{attribute 'linkalways'} 
{attribute 'no_explicit_call' := 'This FB is a CLASS and must be accessed using methods or properties'}
{attribute 'enable_dynamic_creation'}
FUNCTION_BLOCK FINAL MUL_INT EXTENDS Node
VAR
	in1 : _INT(0);
	in2 : _INT(0);
	out : _INT(0);
END_VAR

METHOD PUBLIC Clone : I_Node
VAR
	pNode : POINTER TO MUL_INT;
END_VAR
pNode := __NEW(MUL_INT);
Clone := pNode^;
END_METHOD

METHOD FB_init : BOOL
VAR_INPUT
	bInitRetains : BOOL; // if TRUE, the retain variables are initialized (warm start / cold start)
	bInCopyCode : BOOL;  // if TRUE, the instance afterwards gets moved into the copy code (online change)
END_VAR
AddInput('in1',THIS^.in1);
AddInput('in2',THIS^.in2);
AddOutput('out', THIS^.out);
END_METHOD

METHOD PROTECTED OnExecute
VAR
END_VAR
out.Value := in1.Value * in2.Value;
END_METHOD

END_FUNCTION_BLOCK

(* stored: Version 1.1.0.1, ProductVersion 3.1.4024.15
   POU MUL_INT: Id {147e88f2-4c59-4cc2-a2c0-754993355c72}, SpecialFunc None
   Folder Constructor: Id {3311f08b-3fa3-4e51-8756-cc330fadf173}
   Method Clone: Id {b40a4033-6b0e-495e-9787-c626b4714363}
   Method FB_init: Id {e59e663f-03ca-4856-bd72-29a2773ede71}
   Method OnExecute: Id {e05ddb4e-1e3f-4e19-9133-51f488ba6d44} *)
